{attribute 'qualified_only'}
{attribute 'strict'}
{attribute 'to_string'}
TYPE E_KNXnetIPStateRequest :
(
	eInit 									:= 0,
	eWaitForNextRequest						:= 1
);
END_TYPE

(* stored: Version 1.1.0.1
   DUT E_KNXnetIPStateRequest: Id {dcafb019-88ab-4aa1-93fc-b06d12764590} *)
